// TIA Portal V21 export
FUNCTION "FC604" : Void   // FC604, LAD
TITLE = FC604
{ S7_Optimized_Access := 'TRUE' }
// CIP BLOCK CALL
// stored: AutoNumber false, SetENOAutomatically false
BEGIN

REGION Network 1: #CycleSelection
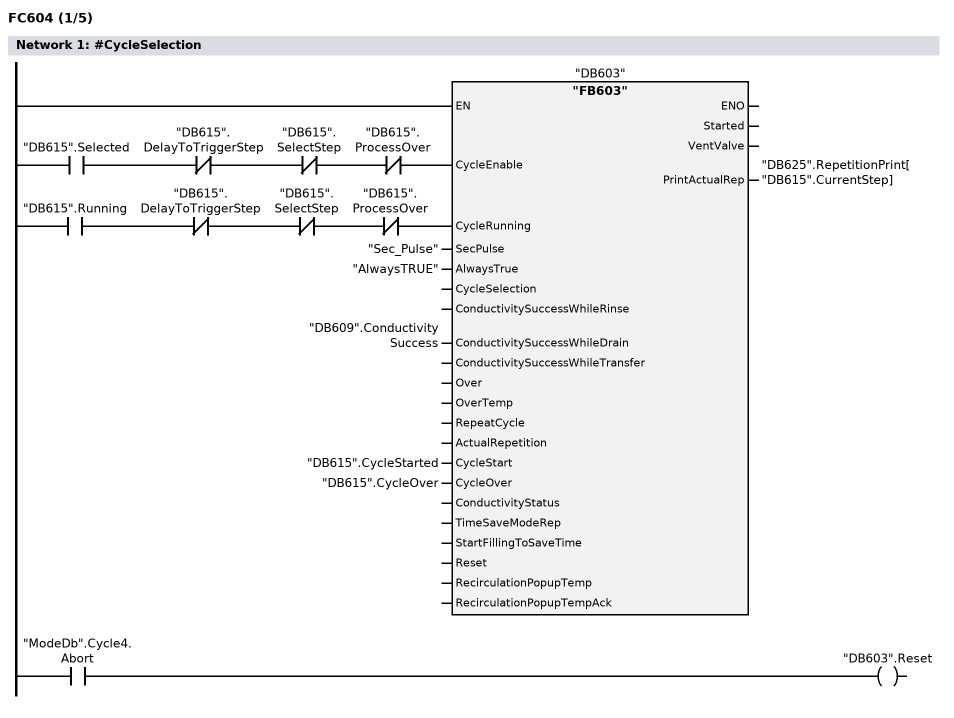
   RUNG wire#powerrail
      "DB603"(CycleEnable := wire#w1, CycleRunning := wire#w2, SecPulse := "Sec_Pulse", AlwaysTrue := "AlwaysTRUE", CycleSelection :=, ConductivitySuccessWhileRinse :=, ConductivitySuccessWhileDrain := "DB609".ConductivitySuccess, ConductivitySuccessWhileTransfer :=, Over :=, OverTemp :=, RepeatCycle :=, ActualRepetition :=, CycleStart := "DB615".CycleStarted, CycleOver := "DB615".CycleOver, ConductivityStatus :=, TimeSaveModeRep :=, StartFillingToSaveTime :=, Reset :=, RecirculationPopupTemp :=, RecirculationPopupTempAck :=, Started =>, VentValve =>, PrintActualRep => "DB625".RepetitionPrint["DB615".CurrentStep])
   END_RUNG
   RUNG wire#powerrail
      Contact( "DB615".Selected )
      I_Contact( "DB615".DelayToTriggerStep )
      I_Contact( "DB615".SelectStep )
      I_Contact( "DB615".ProcessOver )
   END_RUNG wire#w1
   RUNG wire#powerrail
      Contact( "DB615".Running )
      I_Contact( "DB615".DelayToTriggerStep )
      I_Contact( "DB615".SelectStep )
      I_Contact( "DB615".ProcessOver )
   END_RUNG wire#w2
   RUNG wire#powerrail
      Contact( "ModeDb".Cycle4.Abort )
      Coil( "DB603".Reset )
   END_RUNG
   // the same network as SCL:
   "DB603"(CycleEnable := "DB615".Selected AND NOT "DB615".DelayToTriggerStep AND NOT "DB615".SelectStep AND NOT "DB615".ProcessOver,   // "FB603"
           CycleRunning := "DB615".Running AND NOT "DB615".DelayToTriggerStep AND NOT "DB615".SelectStep AND NOT "DB615".ProcessOver,
           SecPulse := "Sec_Pulse",
           AlwaysTrue := "AlwaysTRUE",
           ConductivitySuccessWhileDrain := "DB609".ConductivitySuccess,
           CycleStart := "DB615".CycleStarted,
           CycleOver := "DB615".CycleOver,
           PrintActualRep => "DB625".RepetitionPrint["DB615".CurrentStep]);
   "DB603".Reset := "ModeDb".Cycle4.Abort;
END_REGION

REGION Network 2: #Filling
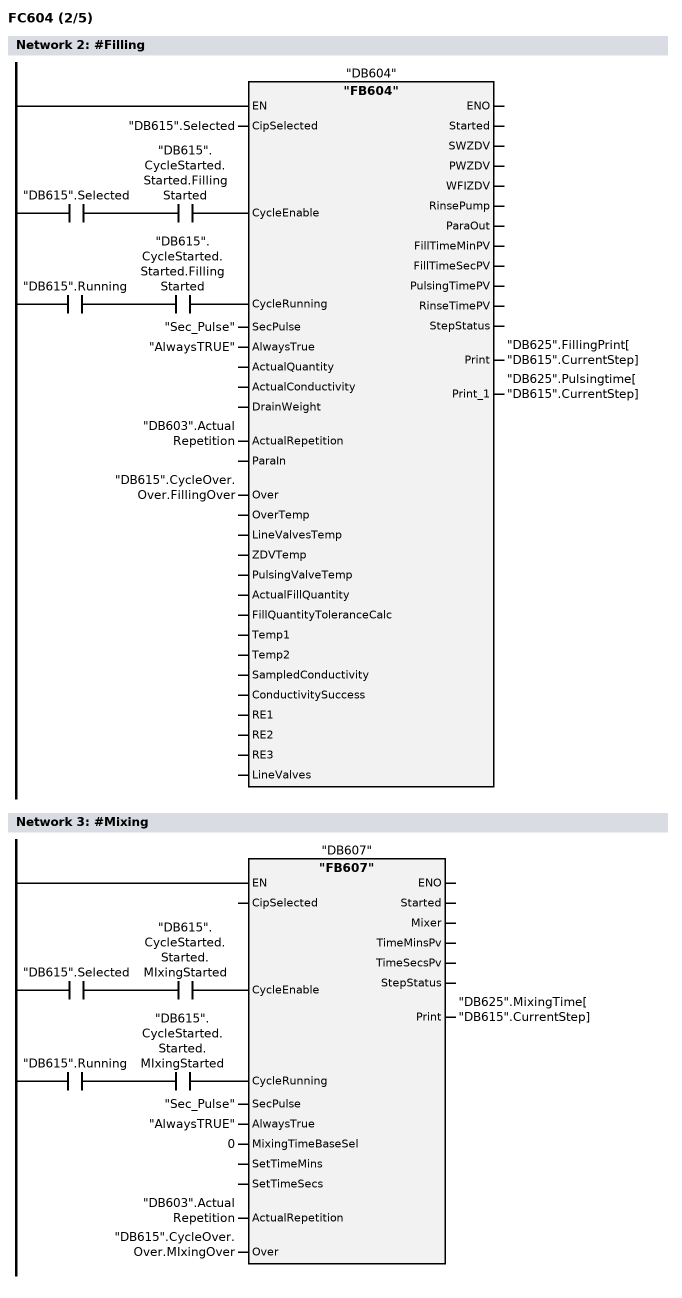
   RUNG wire#powerrail
      "DB604"(CycleEnable := wire#w1, CycleRunning := wire#w2, CipSelected := "DB615".Selected, SecPulse := "Sec_Pulse", AlwaysTrue := "AlwaysTRUE", ActualQuantity :=, ActualConductivity :=, DrainWeight :=, ActualRepetition := "DB603".ActualRepetition, ParaIn :=, Over := "DB615".CycleOver.Over.FillingOver, OverTemp :=, LineValvesTemp :=, ZDVTemp :=, PulsingValveTemp :=, ActualFillQuantity :=, FillQuantityToleranceCalc :=, Temp1 :=, Temp2 :=, SampledConductivity :=, ConductivitySuccess :=, RE1 :=, RE2 :=, RE3 :=, LineValves :=, Started =>, SWZDV =>, PWZDV =>, WFIZDV =>, RinsePump =>, ParaOut =>, FillTimeMinPV =>, FillTimeSecPV =>, PulsingTimePV =>, RinseTimePV =>, StepStatus =>, Print => "DB625".FillingPrint["DB615".CurrentStep], Print_1 => "DB625".Pulsingtime["DB615".CurrentStep])
   END_RUNG
   RUNG wire#powerrail
      Contact( "DB615".Selected )
      Contact( "DB615".CycleStarted.Started.FillingStarted )
   END_RUNG wire#w1
   RUNG wire#powerrail
      Contact( "DB615".Running )
      Contact( "DB615".CycleStarted.Started.FillingStarted )
   END_RUNG wire#w2
   // the same network as SCL:
   "DB604"(CipSelected := "DB615".Selected,   // "FB604"
           CycleEnable := "DB615".Selected AND "DB615".CycleStarted.Started.FillingStarted,
           CycleRunning := "DB615".Running AND "DB615".CycleStarted.Started.FillingStarted,
           SecPulse := "Sec_Pulse",
           AlwaysTrue := "AlwaysTRUE",
           ActualRepetition := "DB603".ActualRepetition,
           Over := "DB615".CycleOver.Over.FillingOver,
           Print => "DB625".FillingPrint["DB615".CurrentStep],
           Print_1 => "DB625".Pulsingtime["DB615".CurrentStep]);
END_REGION

REGION Network 3: #Mixing
   RUNG wire#powerrail
      "DB607"(CycleEnable := wire#w1, CycleRunning := wire#w2, CipSelected :=, SecPulse := "Sec_Pulse", AlwaysTrue := "AlwaysTRUE", MixingTimeBaseSel := 0, SetTimeMins :=, SetTimeSecs :=, ActualRepetition := "DB603".ActualRepetition, Over := "DB615".CycleOver.Over.MIxingOver, Started =>, Mixer =>, TimeMinsPv =>, TimeSecsPv =>, StepStatus =>, Print => "DB625".MixingTime["DB615".CurrentStep])
   END_RUNG
   RUNG wire#powerrail
      Contact( "DB615".Selected )
      Contact( "DB615".CycleStarted.Started.MIxingStarted )
   END_RUNG wire#w1
   RUNG wire#powerrail
      Contact( "DB615".Running )
      Contact( "DB615".CycleStarted.Started.MIxingStarted )
   END_RUNG wire#w2
   // the same network as SCL:
   "DB607"(CycleEnable := "DB615".Selected AND "DB615".CycleStarted.Started.MIxingStarted,   // "FB607"
           CycleRunning := "DB615".Running AND "DB615".CycleStarted.Started.MIxingStarted,
           SecPulse := "Sec_Pulse",
           AlwaysTrue := "AlwaysTRUE",
           MixingTimeBaseSel := 0,
           ActualRepetition := "DB603".ActualRepetition,
           Over := "DB615".CycleOver.Over.MIxingOver,
           Print => "DB625".MixingTime["DB615".CurrentStep]);
END_REGION

REGION Network 4: #Recirculation
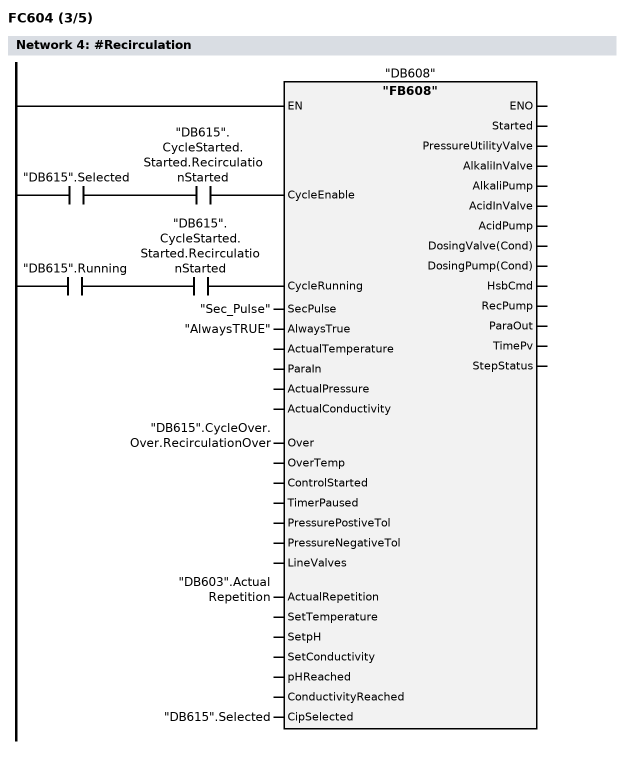
   RUNG wire#powerrail
      "DB608"(CycleEnable := wire#w1, CycleRunning := wire#w2, SecPulse := "Sec_Pulse", AlwaysTrue := "AlwaysTRUE", ActualTemperature :=, ParaIn :=, ActualPressure :=, ActualConductivity :=, Over := "DB615".CycleOver.Over.RecirculationOver, OverTemp :=, ControlStarted :=, TimerPaused :=, PressurePostiveTol :=, PressureNegativeTol :=, LineValves :=, ActualRepetition := "DB603".ActualRepetition, SetTemperature :=, SetpH :=, SetConductivity :=, pHReached :=, ConductivityReached :=, CipSelected := "DB615".Selected, Started =>, PressureUtilityValve =>, AlkaliInValve =>, AlkaliPump =>, AcidInValve =>, AcidPump =>, "DosingValve(Cond)" =>, "DosingPump(Cond)" =>, HsbCmd =>, RecPump =>, ParaOut =>, TimePv =>, StepStatus =>)
   END_RUNG
   RUNG wire#powerrail
      Contact( "DB615".Selected )
      Contact( "DB615".CycleStarted.Started.RecirculationStarted )
   END_RUNG wire#w1
   RUNG wire#powerrail
      Contact( "DB615".Running )
      Contact( "DB615".CycleStarted.Started.RecirculationStarted )
   END_RUNG wire#w2
   // the same network as SCL:
   "DB608"(CycleEnable := "DB615".Selected AND "DB615".CycleStarted.Started.RecirculationStarted,   // "FB608"
           CycleRunning := "DB615".Running AND "DB615".CycleStarted.Started.RecirculationStarted,
           SecPulse := "Sec_Pulse",
           AlwaysTrue := "AlwaysTRUE",
           Over := "DB615".CycleOver.Over.RecirculationOver,
           ActualRepetition := "DB603".ActualRepetition,
           CipSelected := "DB615".Selected);
END_REGION

REGION Network 5: #Drain
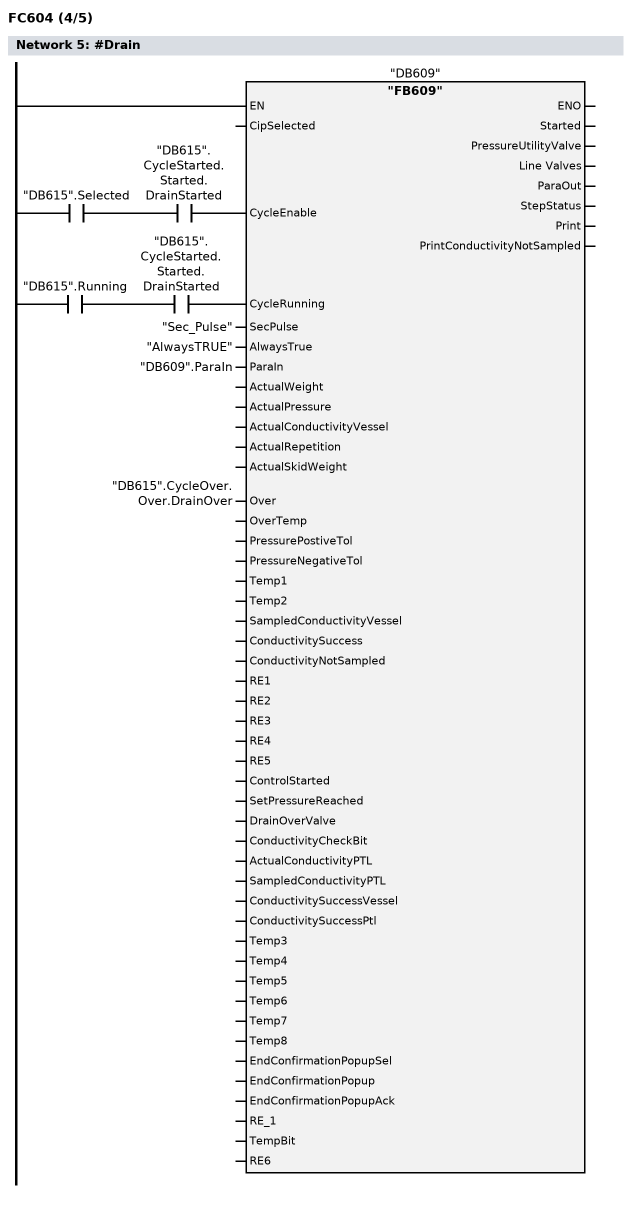
   RUNG wire#powerrail
      "DB609"(CycleEnable := wire#w1, CycleRunning := wire#w2, CipSelected :=, SecPulse := "Sec_Pulse", AlwaysTrue := "AlwaysTRUE", ParaIn := "DB609".ParaIn, ActualWeight :=, ActualPressure :=, ActualConductivityVessel :=, ActualRepetition :=, ActualSkidWeight :=, Over := "DB615".CycleOver.Over.DrainOver, OverTemp :=, PressurePostiveTol :=, PressureNegativeTol :=, Temp1 :=, Temp2 :=, SampledConductivityVessel :=, ConductivitySuccess :=, ConductivityNotSampled :=, RE1 :=, RE2 :=, RE3 :=, RE4 :=, RE5 :=, ControlStarted :=, SetPressureReached :=, DrainOverValve :=, ConductivityCheckBit :=, ActualConductivityPTL :=, SampledConductivityPTL :=, ConductivitySuccessVessel :=, ConductivitySuccessPtl :=, Temp3 :=, Temp4 :=, Temp5 :=, Temp6 :=, Temp7 :=, Temp8 :=, EndConfirmationPopupSel :=, EndConfirmationPopup :=, EndConfirmationPopupAck :=, RE_1 :=, TempBit :=, RE6 :=, Started =>, PressureUtilityValve =>, "Line Valves" =>, ParaOut =>, StepStatus =>, Print =>, PrintConductivityNotSampled =>)
   END_RUNG
   RUNG wire#powerrail
      Contact( "DB615".Selected )
      Contact( "DB615".CycleStarted.Started.DrainStarted )
   END_RUNG wire#w1
   RUNG wire#powerrail
      Contact( "DB615".Running )
      Contact( "DB615".CycleStarted.Started.DrainStarted )
   END_RUNG wire#w2
   // the same network as SCL:
   "DB609"(CycleEnable := "DB615".Selected AND "DB615".CycleStarted.Started.DrainStarted,   // "FB609"
           CycleRunning := "DB615".Running AND "DB615".CycleStarted.Started.DrainStarted,
           SecPulse := "Sec_Pulse",
           AlwaysTrue := "AlwaysTRUE",
           ParaIn := "DB609".ParaIn,
           Over := "DB615".CycleOver.Over.DrainOver);
END_REGION

REGION Network 6: #SystemDrain
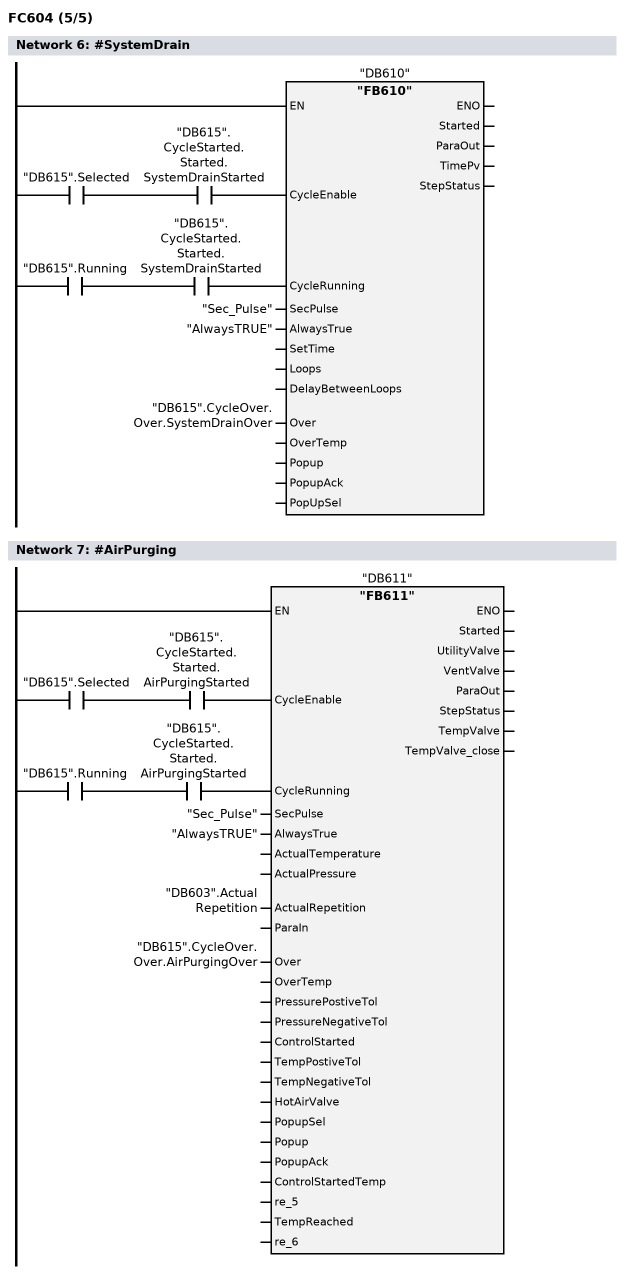
   RUNG wire#powerrail
      "DB610"(CycleEnable := wire#w1, CycleRunning := wire#w2, SecPulse := "Sec_Pulse", AlwaysTrue := "AlwaysTRUE", SetTime :=, Loops :=, DelayBetweenLoops :=, Over := "DB615".CycleOver.Over.SystemDrainOver, OverTemp :=, Popup :=, PopupAck :=, PopUpSel :=, Started =>, ParaOut =>, TimePv =>, StepStatus =>)
   END_RUNG
   RUNG wire#powerrail
      Contact( "DB615".Selected )
      Contact( "DB615".CycleStarted.Started.SystemDrainStarted )
   END_RUNG wire#w1
   RUNG wire#powerrail
      Contact( "DB615".Running )
      Contact( "DB615".CycleStarted.Started.SystemDrainStarted )
   END_RUNG wire#w2
   // the same network as SCL:
   "DB610"(CycleEnable := "DB615".Selected AND "DB615".CycleStarted.Started.SystemDrainStarted,   // "FB610"
           CycleRunning := "DB615".Running AND "DB615".CycleStarted.Started.SystemDrainStarted,
           SecPulse := "Sec_Pulse",
           AlwaysTrue := "AlwaysTRUE",
           Over := "DB615".CycleOver.Over.SystemDrainOver);
END_REGION

REGION Network 7: #AirPurging
   RUNG wire#powerrail
      "DB611"(CycleEnable := wire#w1, CycleRunning := wire#w2, SecPulse := "Sec_Pulse", AlwaysTrue := "AlwaysTRUE", ActualTemperature :=, ActualPressure :=, ActualRepetition := "DB603".ActualRepetition, ParaIn :=, Over := "DB615".CycleOver.Over.AirPurgingOver, OverTemp :=, PressurePostiveTol :=, PressureNegativeTol :=, ControlStarted :=, TempPostiveTol :=, TempNegativeTol :=, HotAirValve :=, PopupSel :=, Popup :=, PopupAck :=, ControlStartedTemp :=, re_5 :=, TempReached :=, re_6 :=, Started =>, UtilityValve =>, VentValve =>, ParaOut =>, StepStatus =>, TempValve =>, TempValve_close =>)
   END_RUNG
   RUNG wire#powerrail
      Contact( "DB615".Selected )
      Contact( "DB615".CycleStarted.Started.AirPurgingStarted )
   END_RUNG wire#w1
   RUNG wire#powerrail
      Contact( "DB615".Running )
      Contact( "DB615".CycleStarted.Started.AirPurgingStarted )
   END_RUNG wire#w2
   // the same network as SCL:
   "DB611"(CycleEnable := "DB615".Selected AND "DB615".CycleStarted.Started.AirPurgingStarted,   // "FB611"
           CycleRunning := "DB615".Running AND "DB615".CycleStarted.Started.AirPurgingStarted,
           SecPulse := "Sec_Pulse",
           AlwaysTrue := "AlwaysTRUE",
           ActualRepetition := "DB603".ActualRepetition,
           Over := "DB615".CycleOver.Over.AirPurgingOver);
END_REGION
END_FUNCTION
